TYPE ST_Places_Inputs :
STRUCT
END_STRUCT
END_TYPE

(* stored: Version 1.1.0.1, ProductVersion 3.1.4024.9
   DUT ST_Places_Inputs: Id {4d3a5405-dd11-47ff-8352-96bdd4158bbb} *)
